# EPICS alarm handler configuration: mps_database/bare/alarms/areas/mpln_ltuh_mp01.alhConfig
GROUP NULL MPLN:LTUH:MP01:1
$ALIAS MPS Link Node 130
$GUIDANCE
LTUH MPS
   Group Name: MPLN:LTUH:MP01:1
   Summary PV:  MPLN:LTUH:MP01:1:STATSUMY
$END
CHANNEL  MPLN:LTUH:MP01:1    MPLN:LTUH:MP01:1:MPS_EN_RBV		-----
CHANNEL  MPLN:LTUH:MP01:1    MPLN:LTUH:MP01:1:LC1_MODE_RBV		-----
